TYPE ST_CommLiftToInfeed :
STRUCT
	bAtInfeedPos : BOOL; // Lift is positioned at the infeed transfer point.
	bReadyForReceiving : BOOL; // Lift is ready to receive a product.
	bProductReceived : BOOL; // Lift confirms product has been received.
END_STRUCT
END_TYPE

(* stored: Version 1.1.0.1, ProductVersion 3.1.4026.13
   DUT ST_CommLiftToInfeed: Id {69a07fb2-ca8a-4689-a717-c131aaa3ba9d} *)
